FUNCTION_BLOCK StateMachineVisitor_Mockup IMPLEMENTS I_ComponentVisitor
VAR
	_StatemachineName : T_MaxString;
END_VAR

PROPERTY StatemachineName : T_MaxString
GET
StatemachineName := _StatemachineName;
END_GET
END_PROPERTY

METHOD VisitComponent
VAR_INPUT
	Component : I_Component;
END_VAR

VAR
	Statemachine : I_Statemachine;
END_VAR
IF __QUERYINTERFACE(Component, Statemachine) THEN
	_StatemachineName := Statemachine.Name;
END_IF
END_METHOD

END_FUNCTION_BLOCK

(* stored: Version 1.1.0.1, ProductVersion 3.1.4026.18
   POU StateMachineVisitor_Mockup: Id {f0911104-906c-4d2b-ab9e-8ff1fbc70401}, SpecialFunc None
   Property StatemachineName: Id {9b49a54f-c2c9-45ca-9ca2-e319cfc86e53}
   Get Get: Id {112992f8-f5e4-4fe7-b1fa-165020a3fe83}
   Method VisitComponent: Id {72bbc9c1-a6bf-40d6-8a45-4816eca45c04} *)
